(* CODESYS project ProfilerLib.library
   Company: Company
   Title: ProfilerLib
   Placeholder: ProfilerLib
   Version: 0.0.0.1

Project tree, tasks and I/O mapping:
  libraries: Tc2_System, * (Beckhoff Automation GmbH)
  Version/
    global variables Global_Version
  function block Profiler [ST]: FB_init, popMethod, pushMethod, setDataRef
  global variables ProfilerParameterList
  data type ProfilerStackStruct
  data type ProfilerStruct
*)

// ProfilerStackStruct
TYPE ProfilerStackStruct :
STRUCT
  hash : UINT;
  depth : DINT;
  startlo : LWORD;
  starthi : LWORD;  
  endlo : LWORD;
  endhi : LWORD;  
END_STRUCT
END_TYPE

// ProfilerStruct
TYPE ProfilerStruct :
STRUCT
  nstack : DINT;
  stacksize : DINT;
  stack : ARRAY[0..ProfilerParameterList.MAX_STACKSIZE] OF ProfilerStackStruct;
  counter : GETCPUCOUNTER;
  enabled : BOOL;
  depth : DINT := 0;   
END_STRUCT
END_TYPE

// Version/Global_Version
{attribute 'TcGenerated'}
// This function has been automatically generated from the project information.
VAR_GLOBAL CONSTANT
	{attribute 'const_non_replaced'}
	{attribute 'linkalways'}
	stLibVersion_ProfilerLib : ST_LibVersion := (iMajor := 0, iMinor := 0, iBuild := 0, iRevision := 1, sVersion := '0.0.0.1');
END_VAR

// ProfilerParameterList
{attribute 'qualified_only'}
VAR_GLOBAL CONSTANT
  MAX_STACKSIZE : DINT := 32000*10;
END_VAR

// Profiler
FUNCTION_BLOCK FINAL Profiler
VAR
  dataRef_ : REFERENCE TO ProfilerStruct;
END_VAR

METHOD FB_init : BOOL
VAR_INPUT
	bInitRetains : BOOL; // if TRUE, the retain variables are initialized (warm start / cold start)
	bInCopyCode : BOOL;  // if TRUE, the instance afterwards gets moved into the copy code (online change)
END_VAR
END_METHOD

METHOD popMethod
VAR_INPUT
  hash : UINT; 
END_VAR
IF NOT __ISVALIDREF(dataRef_)
THEN
  RETURN;
END_IF

IF NOT dataRef_.enabled
THEN
  RETURN;
END_IF

dataRef_.depth := dataRef_.depth - 1;
dataRef_.stack[dataRef_.nstack].depth := dataRef_.depth;
dataRef_.stack[dataRef_.nstack].hash := hash;
dataRef_.stack[dataRef_.nstack].starthi := 0;
dataRef_.stack[dataRef_.nstack].startlo := 0;
dataRef_.counter(cpuCntLoDW => dataRef_.stack[dataRef_.nstack].endlo, cpuCntHiDW => dataRef_.stack[dataRef_.nstack].endhi);

IF dataRef_.depth = 0
THEN
  dataRef_.enabled := FALSE;
  dataRef_.stacksize := dataRef_.nstack;
  dataRef_.nstack := 0;
ELSE
  dataRef_.nstack := dataRef_.nstack + 1;  
END_IF

// abort if the stack is getting too big (too many functions were called)
IF dataRef_.nstack > ProfilerParameterList.MAX_STACKSIZE
THEN
  dataRef_.stacksize := 0;
  dataRef_.enabled := FALSE;
END_IF
END_METHOD

METHOD pushMethod : BOOL
VAR_INPUT
  hash : UINT;  
END_VAR
IF NOT __ISVALIDREF(dataRef_)
THEN
  RETURN;
END_IF

IF NOT dataRef_.enabled
THEN
  RETURN;
END_IF

dataRef_.stack[dataRef_.nstack].depth := dataRef_.depth;
dataRef_.stack[dataRef_.nstack].hash := hash;
dataRef_.counter(cpuCntLoDW => dataRef_.stack[dataRef_.nstack].startlo, cpuCntHiDW => dataRef_.stack[dataRef_.nstack].starthi);
dataRef_.stack[dataRef_.nstack].endhi := 0;
dataRef_.stack[dataRef_.nstack].endlo := 0;
dataRef_.nstack := dataRef_.nstack + 1;
dataRef_.depth := dataRef_.depth + 1;

// abort if the stack is getting too big (too many functions were called)
IF dataRef_.nstack > ProfilerParameterList.MAX_STACKSIZE
THEN
  dataRef_.stacksize := 0;
  dataRef_.enabled := FALSE;
END_IF
END_METHOD

METHOD setDataRef
VAR_INPUT
  dataRef : REFERENCE TO ProfilerStruct;
END_VAR
dataRef_ REF= dataRef;
END_METHOD

END_FUNCTION_BLOCK
